{attribute 'analysis' := '-33'}
// Payload for events
FUNCTION_BLOCK FB_Message
VAR_INPUT
	eLogLevel:			E_LogLevel;
	{attribute 'displaymode':='hex'}
	nID:				UDINT;
	nTimestamp:			Tc2_Utilities.T_FILETIME64;	
	sSource:			STRING(255);
	sType:				STRING(255);
	sMessage:			STRING(255);
	sDefault:			STRING(255);
	sArguments:			STRING(255);
	bActive:			BOOL;
END_VAR
VAR_OUTPUT
END_VAR
VAR
END_VAR
(*
    Tc3_Event – TwinCAT 3 Event Logging Framework
    Copyright (c) Peter Zerlauth

    This component is provided under a Dual Licensing Model:

    1. GPLv3 Open-Source License
       - Free for personal, educational, and non-commercial use.
       - Commercial use allowed only if the entire application is published
         under GPLv3, including all modifications to this code.
       - Requires full disclosure of source code for derivative works.

    2. Commercial License
       - Required for integration into proprietary or closed-source products.
       - Removes all GPLv3 copyleft obligations.
       - Includes optional warranty, professional support, and long-term
         maintenance options.

    For commercial licensing, contact:
        info@peterzerlauth.com

    By using this Function Block you agree to the terms of the selected license.
*)

END_FUNCTION_BLOCK

(* stored: Version 1.1.0.1
   POU FB_Message: Id {84167246-7318-466e-9219-bf236e6d60e2}, SpecialFunc None *)
